FUNCTION_BLOCK FB_OutputNormalizing
VAR_INPUT
	bEnable 			: BOOL;
	fNormalizedInput 	: LREAL;
END_VAR
VAR_OUTPUT
	nOutput 			: INT;
END_VAR
VAR
	nOffset 			: LREAL := 0.0;
	nMaxValue			: LREAL := 32767.0;
	nMinValue 			: LREAL := -32767.0;
	nTempOutput 		: LREAL;
END_VAR


IF fNormalizedInput > 0.0 THEN
	nTempOutput := (fNormalizedInput) * (nMaxValue - nOffset) + nOffset;
ELSIF fNormalizedInput < 0.0 THEN
	nTempOutput := (fNormalizedInput) * (nOffset - nMinValue) + nOffset;
ELSE 
	nTempOutput := nOffset;
END_IF



IF NOT(bEnable) THEN
	nOutput := LREAL_TO_INT(nOffset);
ELSIF (bEnable) THEN
	nOutput := LREAL_TO_INT(nTempOutput);	
END_IF

END_FUNCTION_BLOCK

(* stored: Version 1.1.0.1
   POU FB_OutputNormalizing: Id {c635868d-c90c-4e31-a3e2-f90c8355c566}, SpecialFunc None *)
